# EPICS StreamDevice protocol: bpm.proto
# ./dtwinApp/Db/bpm.proto

Terminator = CR LF;

get_IPM2I00X { out "IPM2I00.XPOS?"; in "IPM2I00.XPOS %f"; ExtraInput = Ignore; }
get_IPM2I00Y { out "IPM2I00.YPOS?"; in "IPM2I00.YPOS %f"; ExtraInput = Ignore; }

get_IPM2I00AX { out "IPM2I00A.XPOS?"; in "IPM2I00A.XPOS %f"; ExtraInput = Ignore; }
get_IPM2I00AY { out "IPM2I00A.YPOS?"; in "IPM2I00A.YPOS %f"; ExtraInput = Ignore; }

get_IPM2I01AX { out "IPM2I01A.XPOS?"; in "IPM2I01A.XPOS %f"; ExtraInput = Ignore; }
get_IPM2I01AY { out "IPM2I01A.YPOS?"; in "IPM2I01A.YPOS %f"; ExtraInput = Ignore; }

get_IPM1I02X { out "IPM1I02.XPOS?"; in "IPM1I02.XPOS %f"; ExtraInput = Ignore; }
get_IPM1I02Y { out "IPM1I02.YPOS?"; in "IPM1I02.YPOS %f"; ExtraInput = Ignore; }

get_IPM1I03X { out "IPM1I03.XPOS?"; in "IPM1I03.XPOS %f"; ExtraInput = Ignore; }
get_IPM1I03Y { out "IPM1I03.YPOS?"; in "IPM1I03.YPOS %f"; ExtraInput = Ignore; }

get_IPM1I04X { out "IPM1I04.XPOS?"; in "IPM1I04.XPOS %f"; ExtraInput = Ignore; }
get_IPM1I04Y { out "IPM1I04.YPOS?"; in "IPM1I04.YPOS %f"; ExtraInput = Ignore; }

get_IPM1I05X { out "IPM1I05.XPOS?"; in "IPM1I05.XPOS %f"; ExtraInput = Ignore; }
get_IPM1I05Y { out "IPM1I05.YPOS?"; in "IPM1I05.YPOS %f"; ExtraInput = Ignore; }

get_IPM1I07X { out "IPM1I07.XPOS?"; in "IPM1I07.XPOS %f"; ExtraInput = Ignore; }
get_IPM1I07Y { out "IPM1I07.YPOS?"; in "IPM1I07.YPOS %f"; ExtraInput = Ignore; }

get_IPM0I01X { out "IPM0I01.XPOS?"; in "IPM0I01.XPOS %f"; ExtraInput = Ignore; }
get_IPM0I01Y { out "IPM0I01.YPOS?"; in "IPM0I01.YPOS %f"; ExtraInput = Ignore; }

get_IPM0I01BX { out "IPM0I01B.XPOS?"; in "IPM0I01B.XPOS %f"; ExtraInput = Ignore; }
get_IPM0I01BY { out "IPM0I01B.YPOS?"; in "IPM0I01B.YPOS %f"; ExtraInput = Ignore; }
